{attribute 'GeneratedUsingTerminal: EL6688-0000-0017'}
{attribute addProperty BoxType "EL6688-0000-0017"}
{attribute addProperty Id "External_SyncAT %I*External_Sync_69535D9824WcStateAT %I*WcState_9091E0EB2InfoDataAT %I*InfoData_1088C70510"}
{attribute addProperty CRC "4246926494"}
{attribute addProperty Size "36"}
TYPE EL6688_FD22F49E EXTENDS EtcSlaveTerminalBase_947E5A46 :
STRUCT
	{attribute addProperty Name "External_Sync"}
	External_Sync : External_Sync_69535D98;
	{attribute addProperty Name "WcState"}
	WcState : WcState_9091E0EB;
	{attribute addProperty Name "InfoData"}
	InfoData : InfoData_1088C705;
END_STRUCT
END_TYPE

(* stored: Version 1.2.0.0, ProductVersion 3.1.4024.9
   DUT EL6688_FD22F49E: Id {824b1e6f-318d-4a3c-a8bf-86bd1b47e652} *)
